TYPE ST_CameraControl :
STRUCT

END_STRUCT
END_TYPE

(* stored: Version 1.1.0.1
   DUT ST_CameraControl: Id {c8ecc2dc-6258-4cc5-a92c-70bda6ad8ec3} *)
